FUNCTION ATAND : LREAL
VAR_INPUT
	TANVAL: LREAL;
END_VAR
VAR
END_VAR

ATAND:=RAD_TO_DEG(ATAN(TANVAL));

END_FUNCTION

(* stored: Version 1.1.0.1, ProductVersion 3.1.4024.12
   POU ATAND: Id {4e832d3b-8433-4700-85c6-a7480922608a}, SpecialFunc None *)
